% RSLogix 500 project LG01815_OriginalPLC_NoTags.RSS, saved by version 12.00.00.00 %
PROJECT "LVD4000"    % processor: MicroLogix 1400 %

PROGRAM FILES
  LAD 2   30 rungs
  LAD 3   3 rungs
  LAD 4   3 rungs
  LAD 5   3 rungs
  LAD 6   3 rungs
  LAD 7   8 rungs
  LAD 8   6 rungs
  LAD 10   21 rungs
  LAD 12   3 rungs
  LAD 14   12 rungs
  LAD 16   24 rungs
  LAD 18   5 rungs
  LAD 20   21 rungs
  LAD 22   2 rungs
  LAD 24   11 rungs
  LAD 26   14 rungs
  LAD 28   19 rungs
  LAD 30   6 rungs
  LAD 32   15 rungs
  LAD 34   20 rungs

DATA FILES
  O0 OUTPUT  6 elements
  I1 INPUT  8 elements
  S2 STATUS  66 elements
  B3 BINARY  256 elements
  T4 TIMER  32 elements
  C5 COUNTER  10 elements
  R6 CONTROL  9 elements
  N7 INTEGER  100 elements
  F8 FLOAT  30 elements
  B9   256 elements
  B11   256 elements
  B12   3 elements
  B14   256 elements
  B15   1 elements
  N16   14 elements
  N17   13 elements
  B18   256 elements
  F19   20 elements
  T20   13 elements
  R21   4 elements
  B22   256 elements
  B23   256 elements
  N24   128 elements
  B25   2 elements

LADDER 2
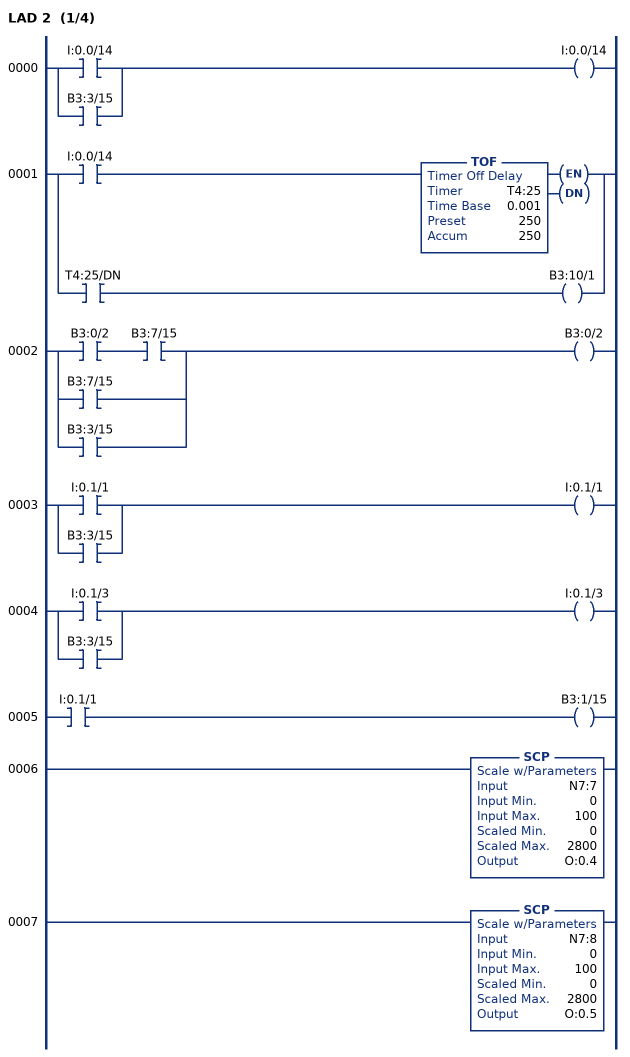
% Rung: 0 %
SOR BST XIC I:0.0/14 NXB XIC B3:3/15 BND OTE I:0.0/14 EOR
% Rung: 1 %
SOR BST XIC I:0.0/14 TOF T4:25 0.001 250 250 NXB XIC T4:25/DN OTE B3:10/1 BND EOR
% Rung: 2 %
SOR BST XIC B3:0/2 XIC B3:7/15 NXB XIC B3:7/15 NXB XIC B3:3/15 BND OTE B3:0/2 EOR
% Rung: 3 %
SOR BST XIC I:0.1/1 NXB XIC B3:3/15 BND OTE I:0.1/1 EOR
% Rung: 4 %
SOR BST XIC I:0.1/3 NXB XIC B3:3/15 BND OTE I:0.1/3 EOR
% Rung: 5 %
SOR XIC I:0.1/1 OTE B3:1/15 EOR
% Rung: 6 %
SOR SCP N7:7 0 100 0 2800 O:0.4 EOR
% Rung: 7 %
SOR SCP N7:8 0 100 0 2800 O:0.5 EOR

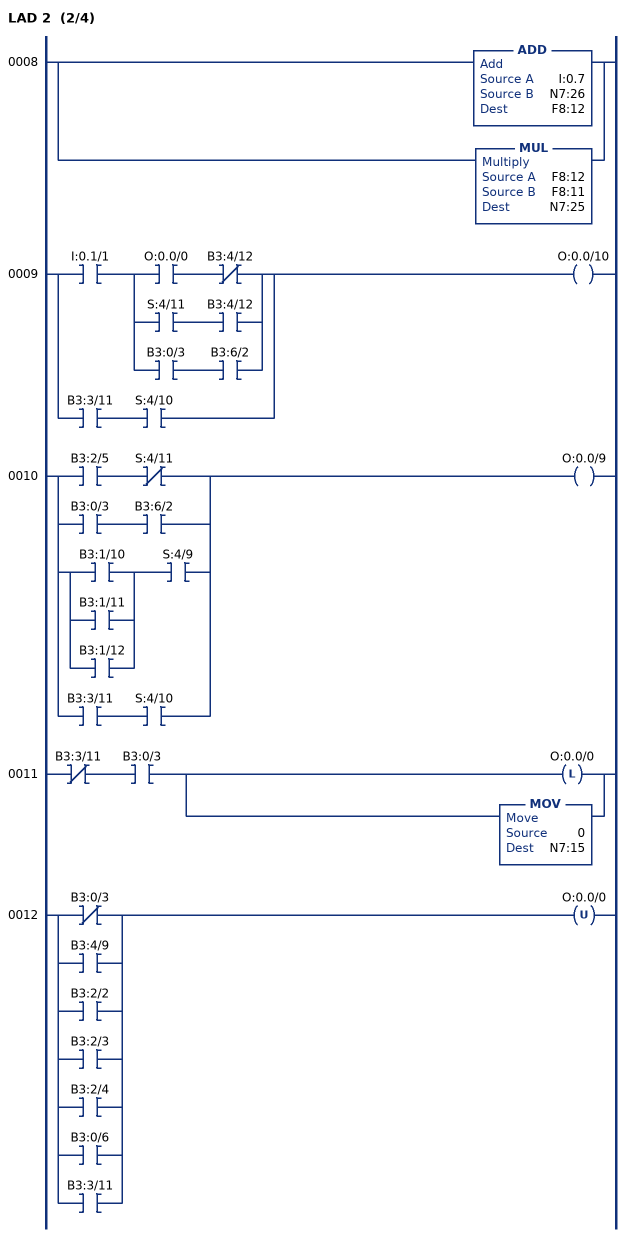
% Rung: 8 %
SOR BST ADD I:0.7 N7:26 F8:12 NXB MUL F8:12 F8:11 N7:25 BND EOR
% Rung: 9 %
SOR BST XIC I:0.1/1 BST XIC O:0.0/0 XIO B3:4/12 NXB XIC S:4/11 XIC B3:4/12 NXB XIC B3:0/3 XIC B3:6/2 BND NXB XIC B3:3/11 XIC S:4/10 BND OTE O:0.0/10 EOR
% Rung: 10 %
SOR BST BST XIC B3:2/5 XIO S:4/11 NXB XIC B3:0/3 XIC B3:6/2 NXB BST XIC B3:1/10 NXB XIC B3:1/11 NXB XIC B3:1/12 BND XIC S:4/9 BND NXB XIC B3:3/11 XIC S:4/10 BND OTE O:0.0/9 EOR
% Rung: 11 %
SOR XIO B3:3/11 XIC B3:0/3 BST OTL O:0.0/0 NXB MOV 0 N7:15 BND EOR
% Rung: 12 %
SOR BST XIO B3:0/3 NXB XIC B3:4/9 NXB XIC B3:2/2 NXB XIC B3:2/3 NXB XIC B3:2/4 NXB XIC B3:0/6 NXB XIC B3:3/11 BND OTU O:0.0/0 EOR

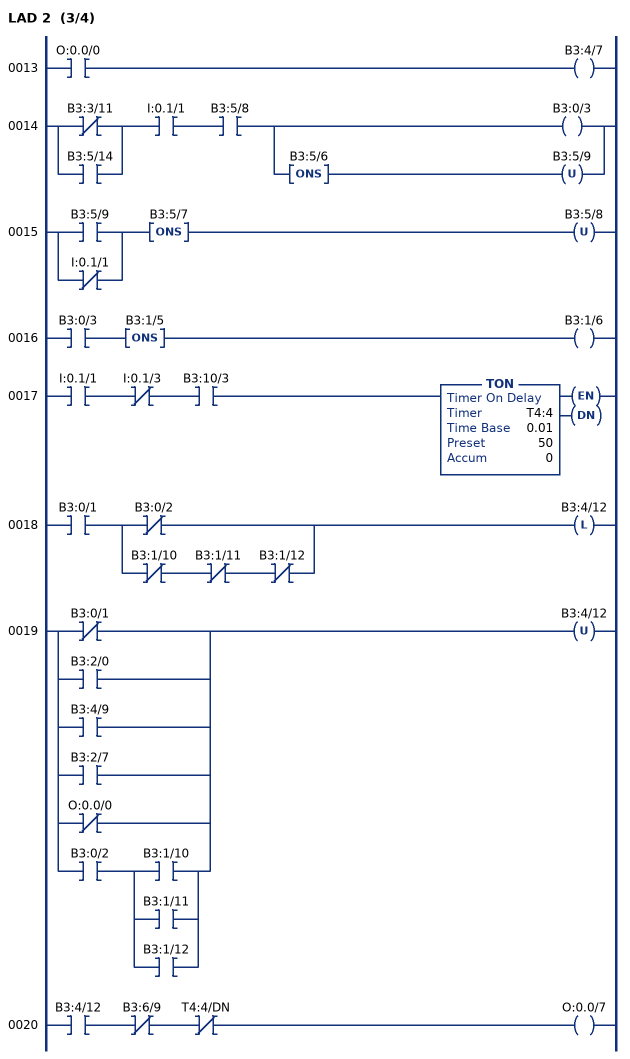
% Rung: 13 %
SOR XIC O:0.0/0 OTE B3:4/7 EOR
% Rung: 14 %
SOR BST XIO B3:3/11 NXB XIC B3:5/14 BND XIC I:0.1/1 XIC B3:5/8 BST OTE B3:0/3 NXB ONS B3:5/6 OTU B3:5/9 BND EOR
% Rung: 15 %
SOR BST XIC B3:5/9 NXB XIO I:0.1/1 BND ONS B3:5/7 OTU B3:5/8 EOR
% Rung: 16 %
SOR XIC B3:0/3 ONS B3:1/5 OTE B3:1/6 EOR
% Rung: 17 %
SOR XIC I:0.1/1 XIO I:0.1/3 XIC B3:10/3 TON T4:4 0.01 50 0 EOR
% Rung: 18 %
SOR XIC B3:0/1 BST XIO B3:0/2 NXB XIO B3:1/10 XIO B3:1/11 XIO B3:1/12 BND OTL B3:4/12 EOR
% Rung: 19 %
SOR BST XIO B3:0/1 NXB XIC B3:2/0 NXB XIC B3:4/9 NXB XIC B3:2/7 NXB XIO O:0.0/0 NXB XIC B3:0/2 BST XIC B3:1/10 NXB XIC B3:1/11 NXB XIC B3:1/12 BND BND OTU B3:4/12 EOR
% Rung: 20 %
SOR XIC B3:4/12 XIO B3:6/9 XIO T4:4/DN OTE O:0.0/7 EOR

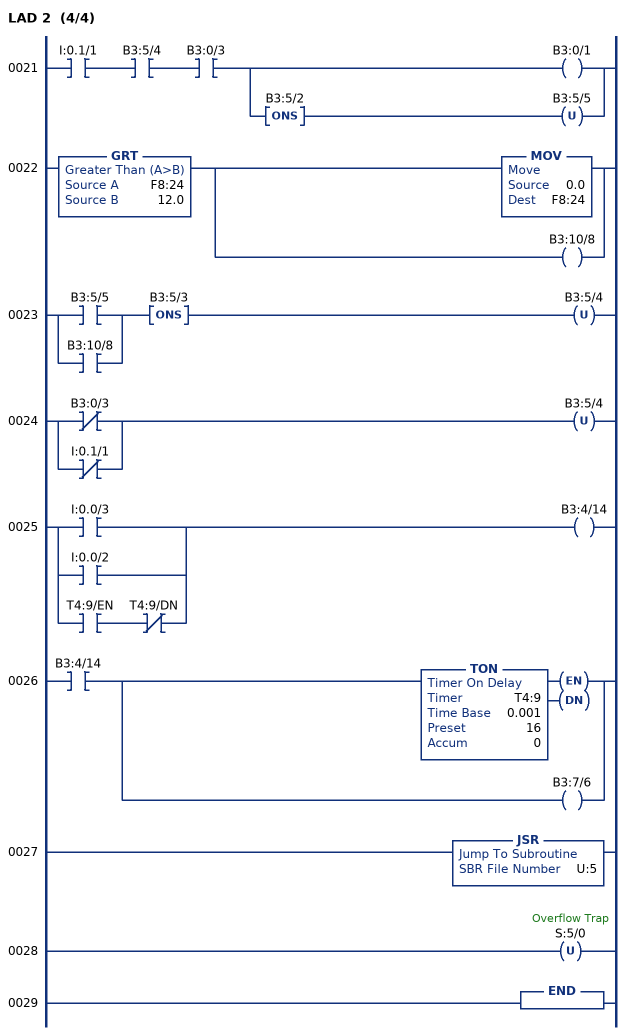
% Rung: 21 %
SOR XIC I:0.1/1 XIC B3:5/4 XIC B3:0/3 BST OTE B3:0/1 NXB ONS B3:5/2 OTU B3:5/5 BND EOR
% Rung: 22 %
SOR GRT F8:24 12.0 BST MOV 0.0 F8:24 NXB OTE B3:10/8 BND EOR
% Rung: 23 %
SOR BST XIC B3:5/5 NXB XIC B3:10/8 BND ONS B3:5/3 OTU B3:5/4 EOR
% Rung: 24 %
SOR BST XIO B3:0/3 NXB XIO I:0.1/1 BND OTU B3:5/4 EOR
% Rung: 25 %
SOR BST XIC I:0.0/3 NXB XIC I:0.0/2 NXB XIC T4:9/EN XIO T4:9/DN BND OTE B3:4/14 EOR
% Rung: 26 %
SOR XIC B3:4/14 BST TON T4:9 0.001 16 0 NXB OTE B3:7/6 BND EOR
% Rung: 27 %
SOR JSR U:5 EOR
% Rung: 28 %
SOR OTU S:5/0 EOR
%   S:5/0  "Overflow Trap" %
% Rung: 29 %
SOR END EOR

LADDER 3
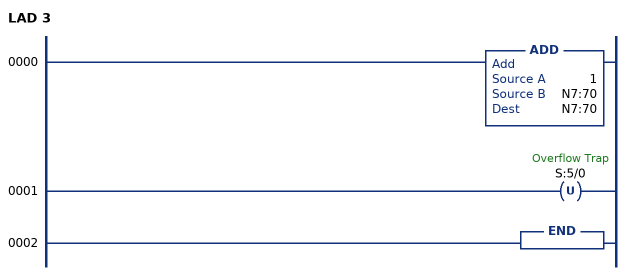
% Rung: 0 %
SOR ADD 1 N7:70 N7:70 EOR
% Rung: 1 %
SOR OTU S:5/0 EOR
%   S:5/0  "Overflow Trap" %
% Rung: 2 %
SOR END EOR

LADDER 4
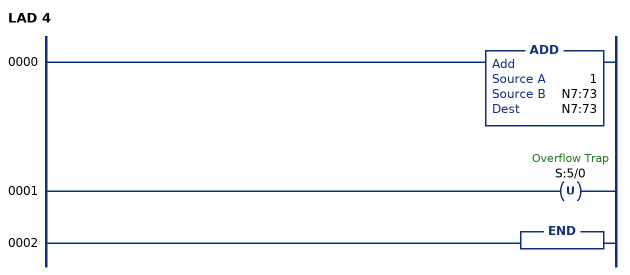
% Rung: 0 %
SOR ADD 1 N7:73 N7:73 EOR
% Rung: 1 %
SOR OTU S:5/0 EOR
%   S:5/0  "Overflow Trap" %
% Rung: 2 %
SOR END EOR

LADDER 5
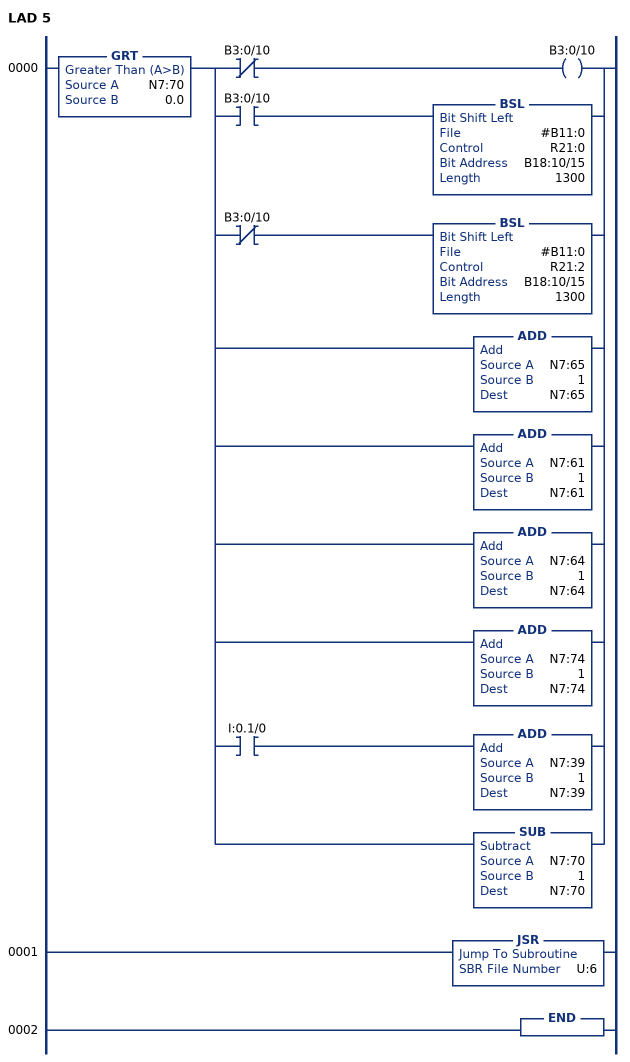
% Rung: 0 %
SOR GRT N7:70 0.0 BST XIO B3:0/10 OTE B3:0/10 NXB XIC B3:0/10 BSL #B11:0 R21:0 B18:10/15 1300 NXB XIO B3:0/10 BSL #B11:0 R21:2 B18:10/15 1300 NXB ADD N7:65 1 N7:65 NXB ADD N7:61 1 N7:61 NXB ADD N7:64 1 N7:64 NXB ADD N7:74 1 N7:74 NXB XIC I:0.1/0 ADD N7:39 1 N7:39 NXB SUB N7:70 1 N7:70 BND EOR
% Rung: 1 %
SOR JSR U:6 EOR
% Rung: 2 %
SOR END EOR

LADDER 6
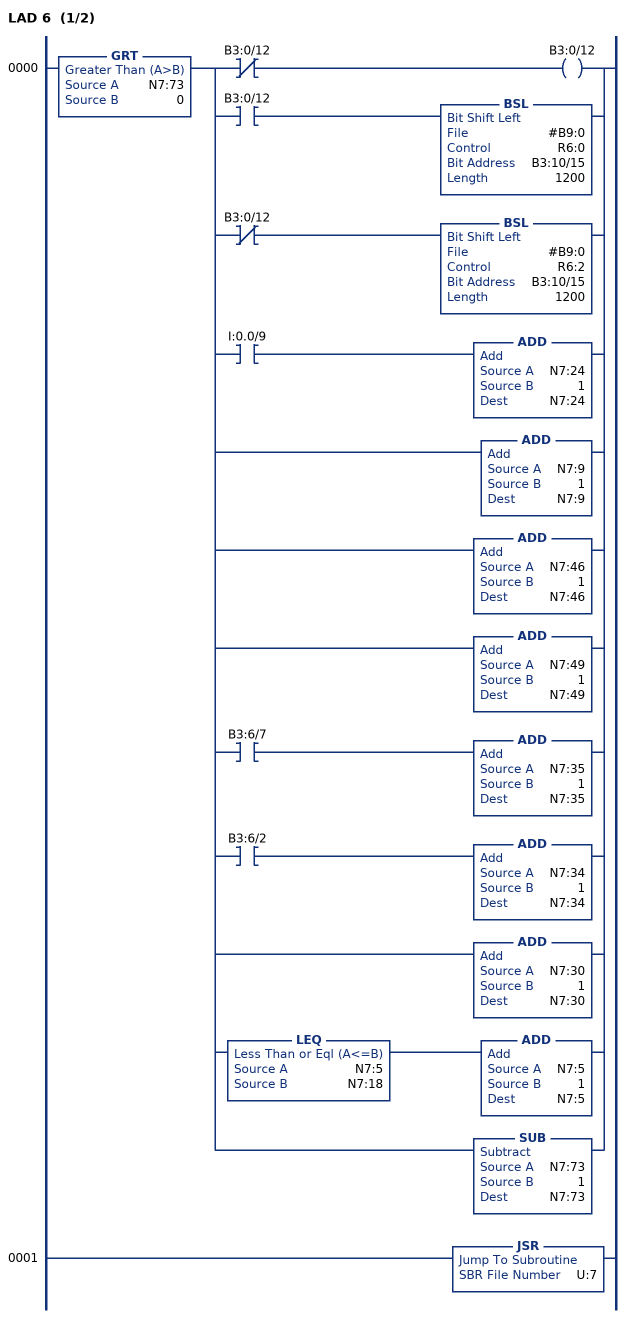
% Rung: 0 %
SOR GRT N7:73 0 BST XIO B3:0/12 OTE B3:0/12 NXB XIC B3:0/12 BSL #B9:0 R6:0 B3:10/15 1200 NXB XIO B3:0/12 BSL #B9:0 R6:2 B3:10/15 1200 NXB XIC I:0.0/9 ADD N7:24 1 N7:24 NXB ADD N7:9 1 N7:9 NXB ADD N7:46 1 N7:46 NXB ADD N7:49 1 N7:49 NXB XIC B3:6/7 ADD N7:35 1 N7:35 NXB XIC B3:6/2 ADD N7:34 1 N7:34 NXB ADD N7:30 1 N7:30 NXB LEQ N7:5 N7:18 ADD N7:5 1 N7:5 NXB SUB N7:73 1 N7:73 BND EOR
% Rung: 1 %
SOR JSR U:7 EOR

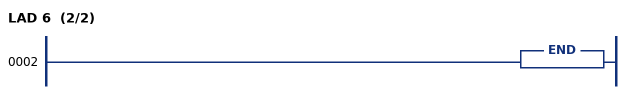
% Rung: 2 %
SOR END EOR

LADDER 7
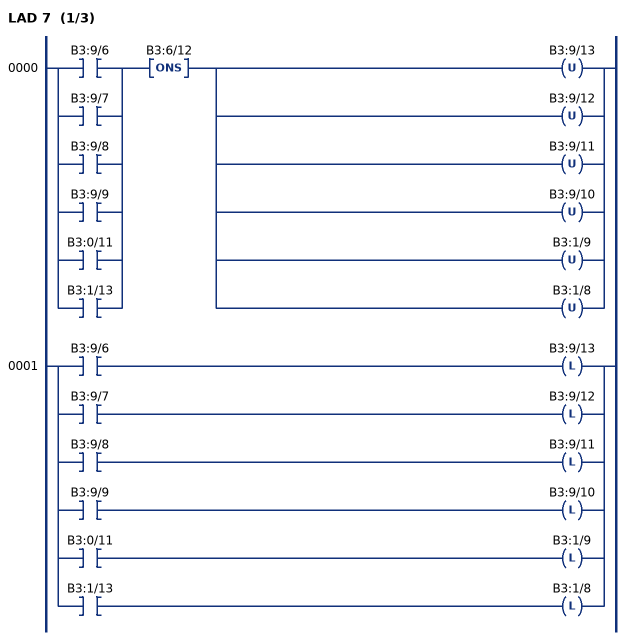
% Rung: 0 %
SOR BST XIC B3:9/6 NXB XIC B3:9/7 NXB XIC B3:9/8 NXB XIC B3:9/9 NXB XIC B3:0/11 NXB XIC B3:1/13 BND ONS B3:6/12 BST OTU B3:9/13 NXB OTU B3:9/12 NXB OTU B3:9/11 NXB OTU B3:9/10 NXB OTU B3:1/9 NXB OTU B3:1/8 BND EOR
% Rung: 1 %
SOR BST XIC B3:9/6 OTL B3:9/13 NXB XIC B3:9/7 OTL B3:9/12 NXB XIC B3:9/8 OTL B3:9/11 NXB XIC B3:9/9 OTL B3:9/10 NXB XIC B3:0/11 OTL B3:1/9 NXB XIC B3:1/13 OTL B3:1/8 BND EOR

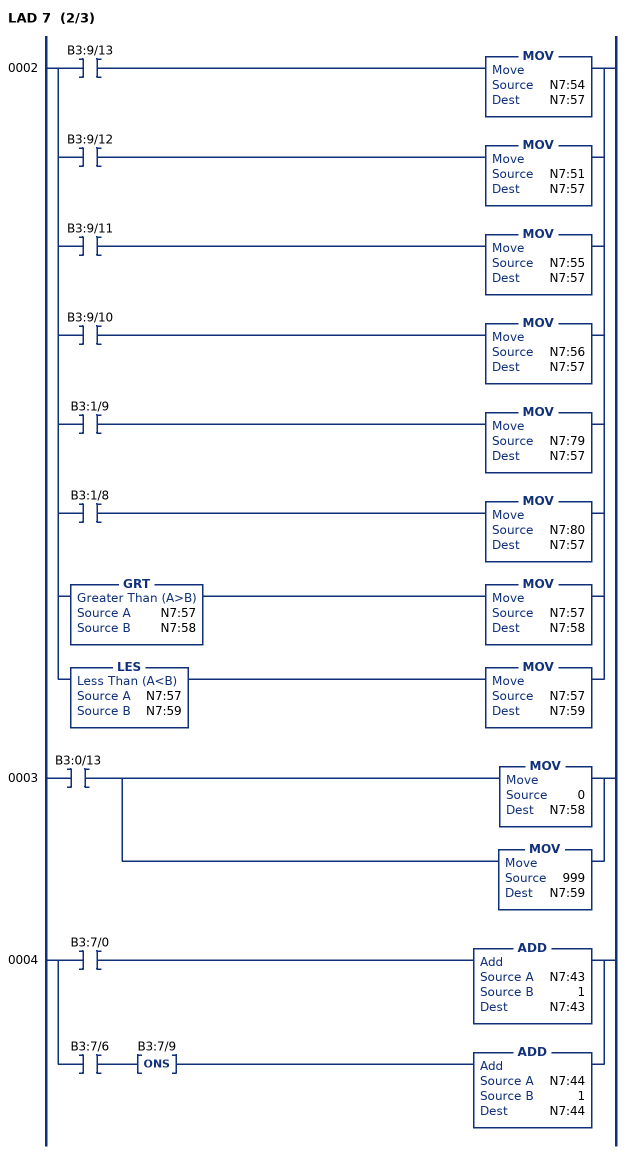
% Rung: 2 %
SOR BST XIC B3:9/13 MOV N7:54 N7:57 NXB XIC B3:9/12 MOV N7:51 N7:57 NXB XIC B3:9/11 MOV N7:55 N7:57 NXB XIC B3:9/10 MOV N7:56 N7:57 NXB XIC B3:1/9 MOV N7:79 N7:57 NXB XIC B3:1/8 MOV N7:80 N7:57 NXB GRT N7:57 N7:58 MOV N7:57 N7:58 NXB LES N7:57 N7:59 MOV N7:57 N7:59 BND EOR
% Rung: 3 %
SOR XIC B3:0/13 BST MOV 0 N7:58 NXB MOV 999 N7:59 BND EOR
% Rung: 4 %
SOR BST XIC B3:7/0 ADD N7:43 1 N7:43 NXB XIC B3:7/6 ONS B3:7/9 ADD N7:44 1 N7:44 BND EOR

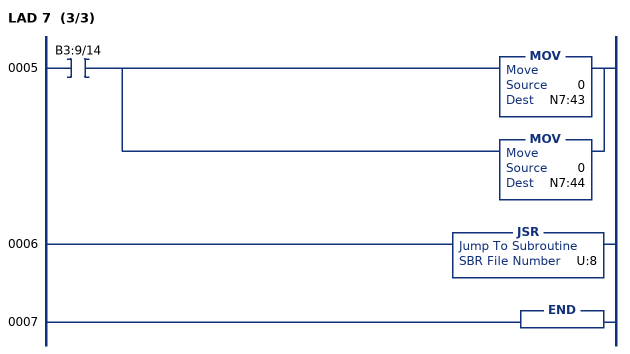
% Rung: 5 %
SOR XIC B3:9/14 BST MOV 0 N7:43 NXB MOV 0 N7:44 BND EOR
% Rung: 6 %
SOR JSR U:8 EOR
% Rung: 7 %
SOR END EOR

LADDER 8
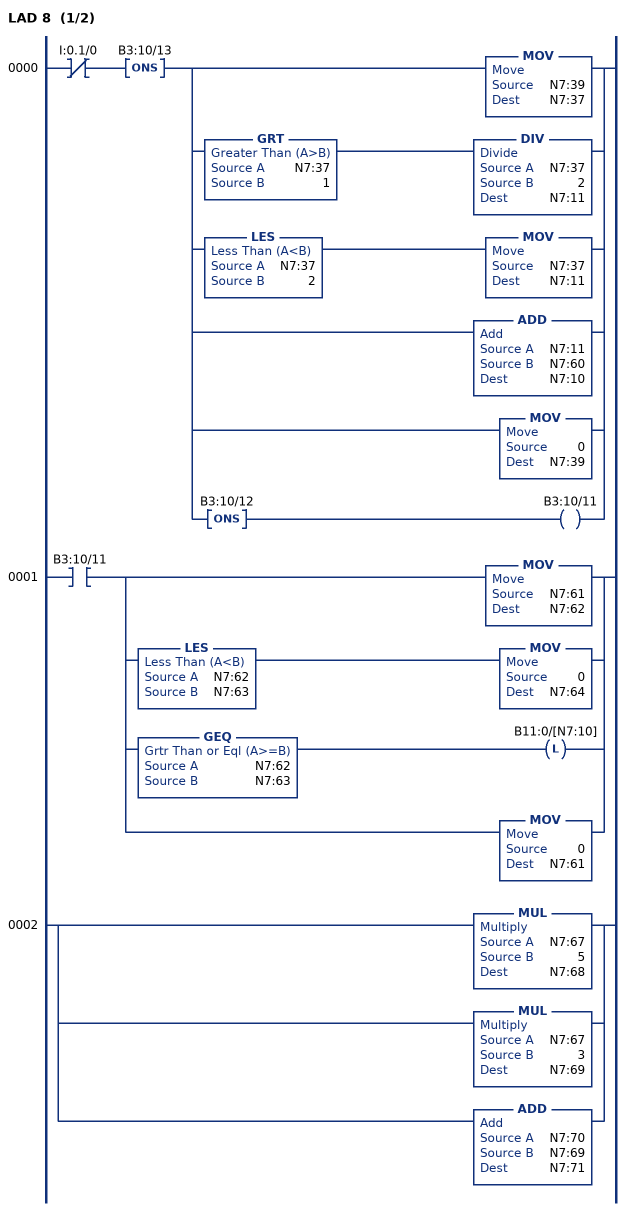
% Rung: 0 %
SOR XIO I:0.1/0 ONS B3:10/13 BST MOV N7:39 N7:37 NXB GRT N7:37 1 DIV N7:37 2 N7:11 NXB LES N7:37 2 MOV N7:37 N7:11 NXB ADD N7:11 N7:60 N7:10 NXB MOV 0 N7:39 NXB ONS B3:10/12 OTE B3:10/11 BND EOR
% Rung: 1 %
SOR XIC B3:10/11 BST MOV N7:61 N7:62 NXB LES N7:62 N7:63 MOV 0 N7:64 NXB GEQ N7:62 N7:63 OTL B11:0/[N7:10] NXB MOV 0 N7:61 BND EOR
% Rung: 2 %
SOR BST MUL N7:67 5 N7:68 NXB MUL N7:67 3 N7:69 NXB ADD N7:70 N7:69 N7:71 BND EOR

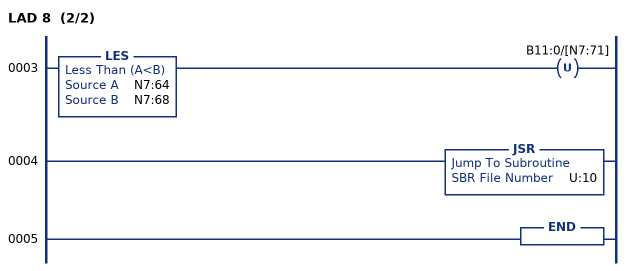
% Rung: 3 %
SOR LES N7:64 N7:68 OTU B11:0/[N7:71] EOR
% Rung: 4 %
SOR JSR U:10 EOR
% Rung: 5 %
SOR END EOR

LADDER 10
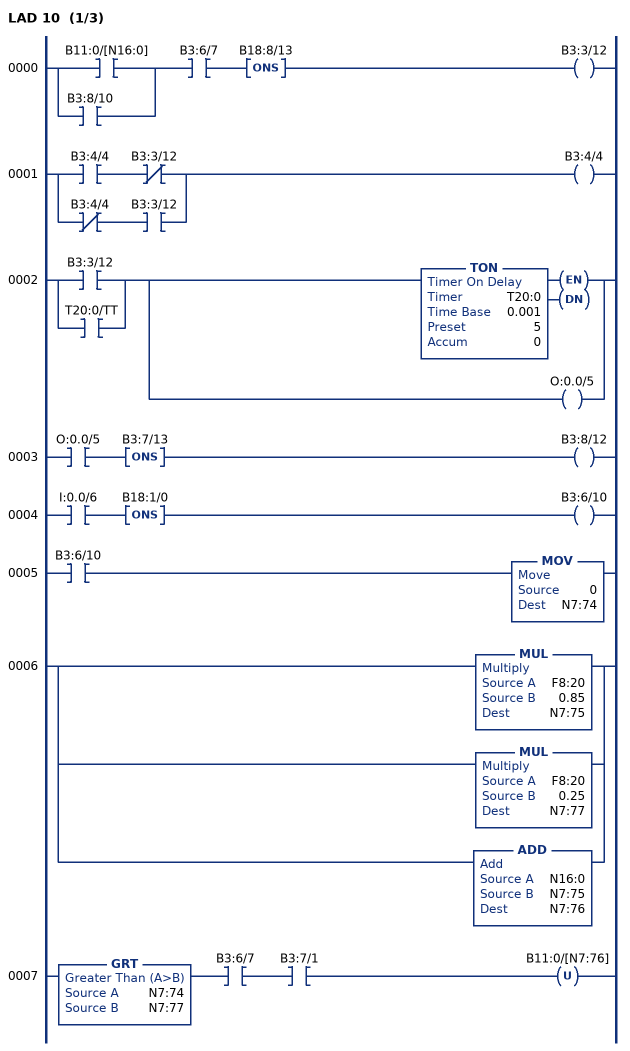
% Rung: 0 %
SOR BST XIC B11:0/[N16:0] NXB XIC B3:8/10 BND XIC B3:6/7 ONS B18:8/13 OTE B3:3/12 EOR
% Rung: 1 %
SOR BST XIC B3:4/4 XIO B3:3/12 NXB XIO B3:4/4 XIC B3:3/12 BND OTE B3:4/4 EOR
% Rung: 2 %
SOR BST XIC B3:3/12 NXB XIC T20:0/TT BND BST TON T20:0 0.001 5 0 NXB OTE O:0.0/5 BND EOR
% Rung: 3 %
SOR XIC O:0.0/5 ONS B3:7/13 OTE B3:8/12 EOR
% Rung: 4 %
SOR XIC I:0.0/6 ONS B18:1/0 OTE B3:6/10 EOR
% Rung: 5 %
SOR XIC B3:6/10 MOV 0 N7:74 EOR
% Rung: 6 %
SOR BST MUL F8:20 0.85 N7:75 NXB MUL F8:20 0.25 N7:77 NXB ADD N16:0 N7:75 N7:76 BND EOR
% Rung: 7 %
SOR GRT N7:74 N7:77 XIC B3:6/7 XIC B3:7/1 OTU B11:0/[N7:76] EOR

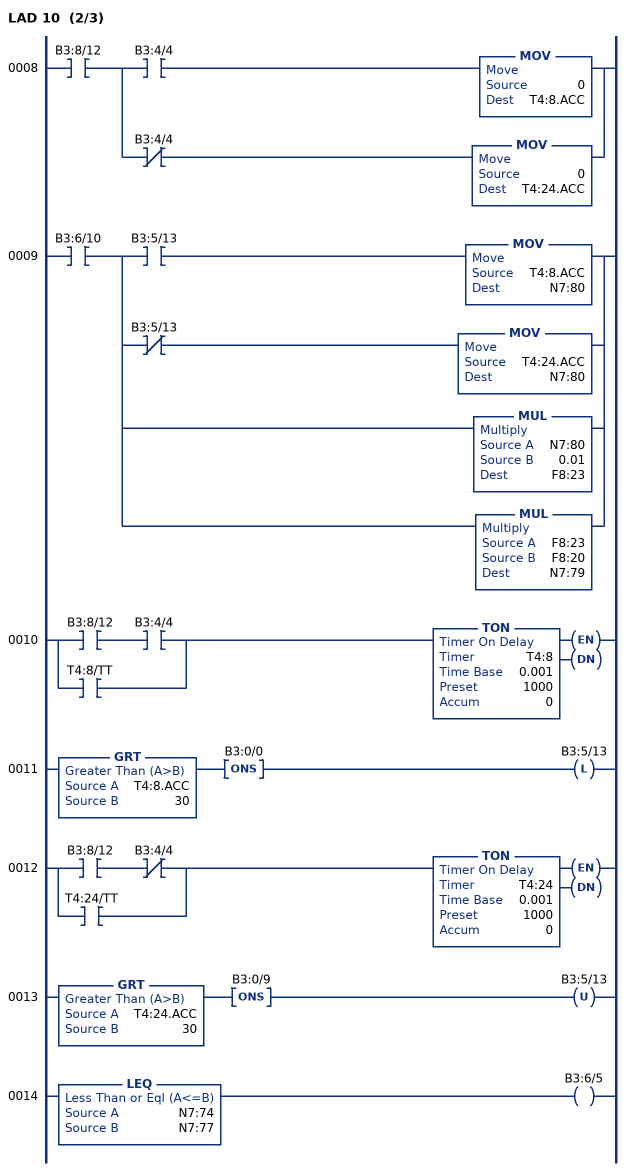
% Rung: 8 %
SOR XIC B3:8/12 BST XIC B3:4/4 MOV 0 T4:8.ACC NXB XIO B3:4/4 MOV 0 T4:24.ACC BND EOR
% Rung: 9 %
SOR XIC B3:6/10 BST XIC B3:5/13 MOV T4:8.ACC N7:80 NXB XIO B3:5/13 MOV T4:24.ACC N7:80 NXB MUL N7:80 0.01 F8:23 NXB MUL F8:23 F8:20 N7:79 BND EOR
% Rung: 10 %
SOR BST XIC B3:8/12 XIC B3:4/4 NXB XIC T4:8/TT BND TON T4:8 0.001 1000 0 EOR
% Rung: 11 %
SOR GRT T4:8.ACC 30 ONS B3:0/0 OTL B3:5/13 EOR
% Rung: 12 %
SOR BST XIC B3:8/12 XIO B3:4/4 NXB XIC T4:24/TT BND TON T4:24 0.001 1000 0 EOR
% Rung: 13 %
SOR GRT T4:24.ACC 30 ONS B3:0/9 OTU B3:5/13 EOR
% Rung: 14 %
SOR LEQ N7:74 N7:77 OTE B3:6/5 EOR

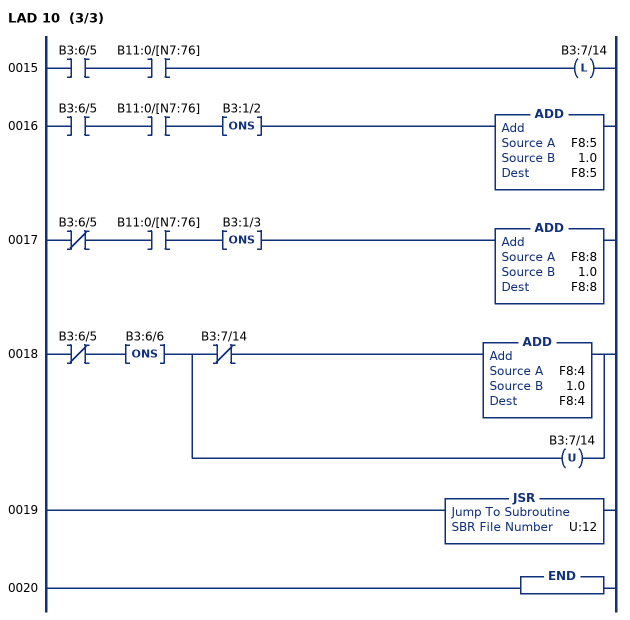
% Rung: 15 %
SOR XIC B3:6/5 XIC B11:0/[N7:76] OTL B3:7/14 EOR
% Rung: 16 %
SOR XIC B3:6/5 XIC B11:0/[N7:76] ONS B3:1/2 ADD F8:5 1.0 F8:5 EOR
% Rung: 17 %
SOR XIO B3:6/5 XIC B11:0/[N7:76] ONS B3:1/3 ADD F8:8 1.0 F8:8 EOR
% Rung: 18 %
SOR XIO B3:6/5 ONS B3:6/6 BST XIO B3:7/14 ADD F8:4 1.0 F8:4 NXB OTU B3:7/14 BND EOR
% Rung: 19 %
SOR JSR U:12 EOR
% Rung: 20 %
SOR END EOR

LADDER 12
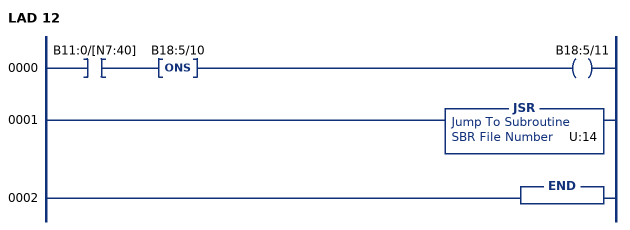
% Rung: 0 %
SOR XIC B11:0/[N7:40] ONS B18:5/10 OTE B18:5/11 EOR
% Rung: 1 %
SOR JSR U:14 EOR
% Rung: 2 %
SOR END EOR

LADDER 14
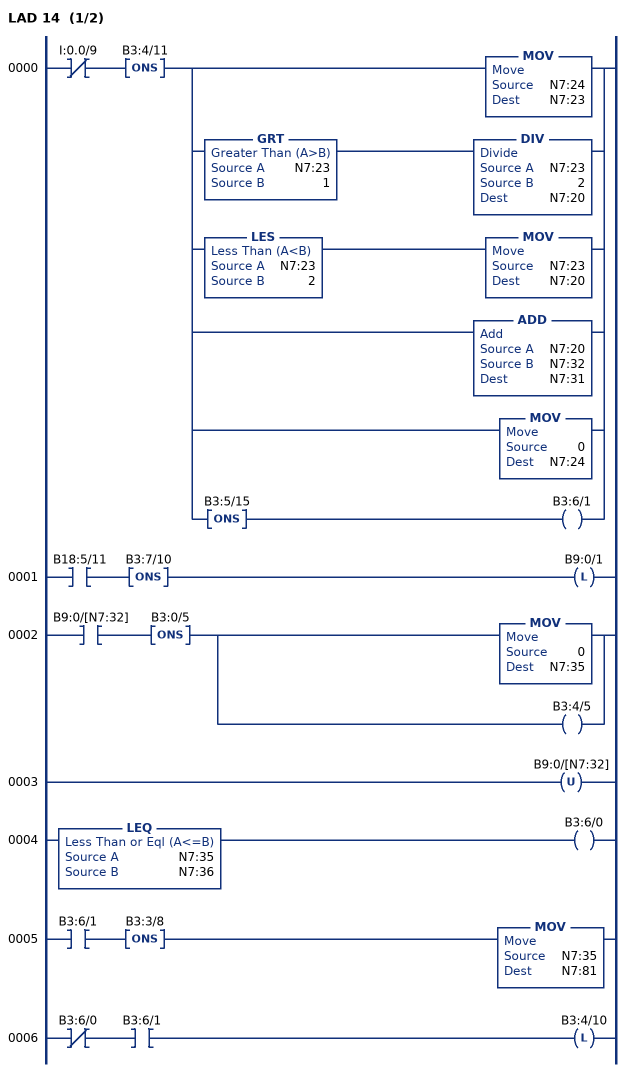
% Rung: 0 %
SOR XIO I:0.0/9 ONS B3:4/11 BST MOV N7:24 N7:23 NXB GRT N7:23 1 DIV N7:23 2 N7:20 NXB LES N7:23 2 MOV N7:23 N7:20 NXB ADD N7:20 N7:32 N7:31 NXB MOV 0 N7:24 NXB ONS B3:5/15 OTE B3:6/1 BND EOR
% Rung: 1 %
SOR XIC B18:5/11 ONS B3:7/10 OTL B9:0/1 EOR
% Rung: 2 %
SOR XIC B9:0/[N7:32] ONS B3:0/5 BST MOV 0 N7:35 NXB OTE B3:4/5 BND EOR
% Rung: 3 %
SOR OTU B9:0/[N7:32] EOR
% Rung: 4 %
SOR LEQ N7:35 N7:36 OTE B3:6/0 EOR
% Rung: 5 %
SOR XIC B3:6/1 ONS B3:3/8 MOV N7:35 N7:81 EOR
% Rung: 6 %
SOR XIO B3:6/0 XIC B3:6/1 OTL B3:4/10 EOR

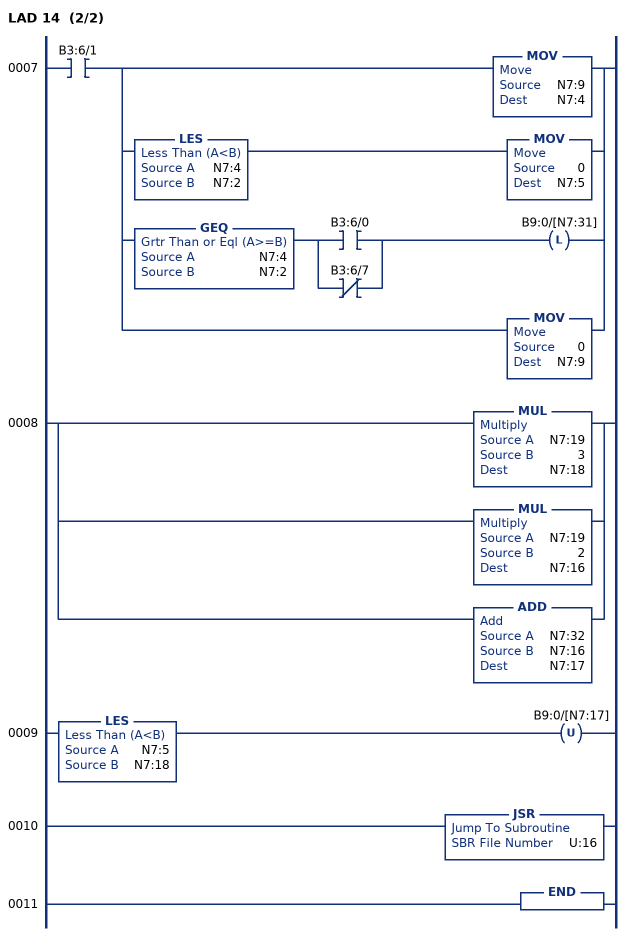
% Rung: 7 %
SOR XIC B3:6/1 BST MOV N7:9 N7:4 NXB LES N7:4 N7:2 MOV 0 N7:5 NXB GEQ N7:4 N7:2 BST XIC B3:6/0 NXB XIO B3:6/7 BND OTL B9:0/[N7:31] NXB MOV 0 N7:9 BND EOR
% Rung: 8 %
SOR BST MUL N7:19 3 N7:18 NXB MUL N7:19 2 N7:16 NXB ADD N7:32 N7:16 N7:17 BND EOR
% Rung: 9 %
SOR LES N7:5 N7:18 OTU B9:0/[N7:17] EOR
% Rung: 10 %
SOR JSR U:16 EOR
% Rung: 11 %
SOR END EOR

LADDER 16
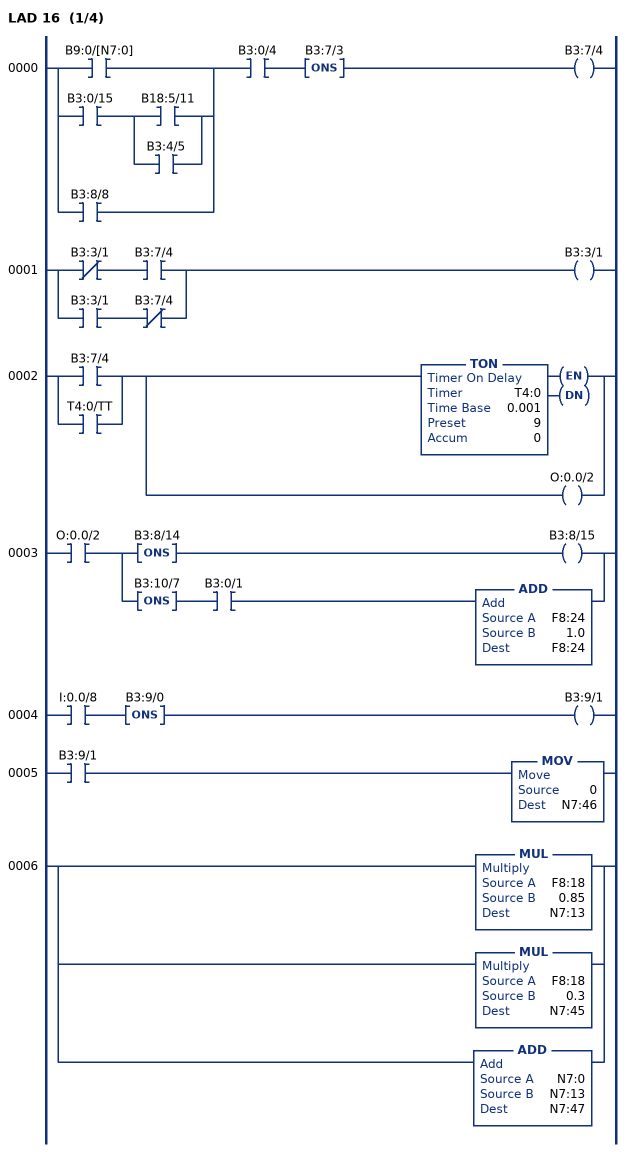
% Rung: 0 %
SOR BST XIC B9:0/[N7:0] NXB XIC B3:0/15 BST XIC B18:5/11 NXB XIC B3:4/5 BND NXB XIC B3:8/8 BND XIC B3:0/4 ONS B3:7/3 OTE B3:7/4 EOR
% Rung: 1 %
SOR BST XIO B3:3/1 XIC B3:7/4 NXB XIC B3:3/1 XIO B3:7/4 BND OTE B3:3/1 EOR
% Rung: 2 %
SOR BST XIC B3:7/4 NXB XIC T4:0/TT BND BST TON T4:0 0.001 9 0 NXB OTE O:0.0/2 BND EOR
% Rung: 3 %
SOR XIC O:0.0/2 BST ONS B3:8/14 OTE B3:8/15 NXB ONS B3:10/7 XIC B3:0/1 ADD F8:24 1.0 F8:24 BND EOR
% Rung: 4 %
SOR XIC I:0.0/8 ONS B3:9/0 OTE B3:9/1 EOR
% Rung: 5 %
SOR XIC B3:9/1 MOV 0 N7:46 EOR
% Rung: 6 %
SOR BST MUL F8:18 0.85 N7:13 NXB MUL F8:18 0.3 N7:45 NXB ADD N7:0 N7:13 N7:47 BND EOR

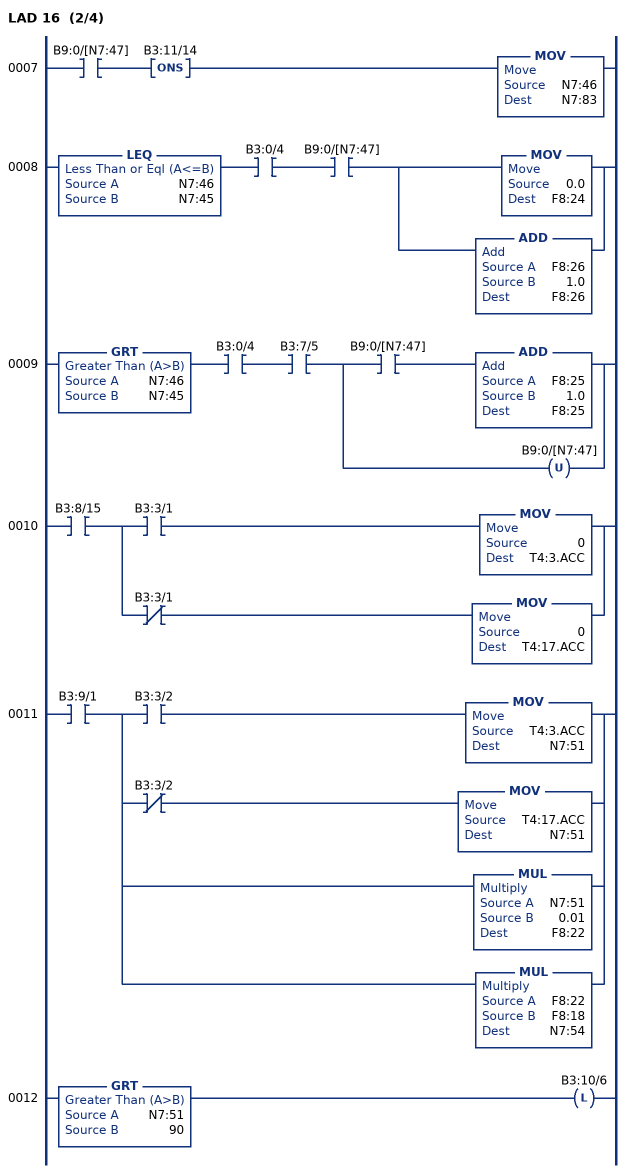
% Rung: 7 %
SOR XIC B9:0/[N7:47] ONS B3:11/14 MOV N7:46 N7:83 EOR
% Rung: 8 %
SOR LEQ N7:46 N7:45 XIC B3:0/4 XIC B9:0/[N7:47] BST MOV 0.0 F8:24 NXB ADD F8:26 1.0 F8:26 BND EOR
% Rung: 9 %
SOR GRT N7:46 N7:45 XIC B3:0/4 XIC B3:7/5 BST XIC B9:0/[N7:47] ADD F8:25 1.0 F8:25 NXB OTU B9:0/[N7:47] BND EOR
% Rung: 10 %
SOR XIC B3:8/15 BST XIC B3:3/1 MOV 0 T4:3.ACC NXB XIO B3:3/1 MOV 0 T4:17.ACC BND EOR
% Rung: 11 %
SOR XIC B3:9/1 BST XIC B3:3/2 MOV T4:3.ACC N7:51 NXB XIO B3:3/2 MOV T4:17.ACC N7:51 NXB MUL N7:51 0.01 F8:22 NXB MUL F8:22 F8:18 N7:54 BND EOR
% Rung: 12 %
SOR GRT N7:51 90 OTL B3:10/6 EOR

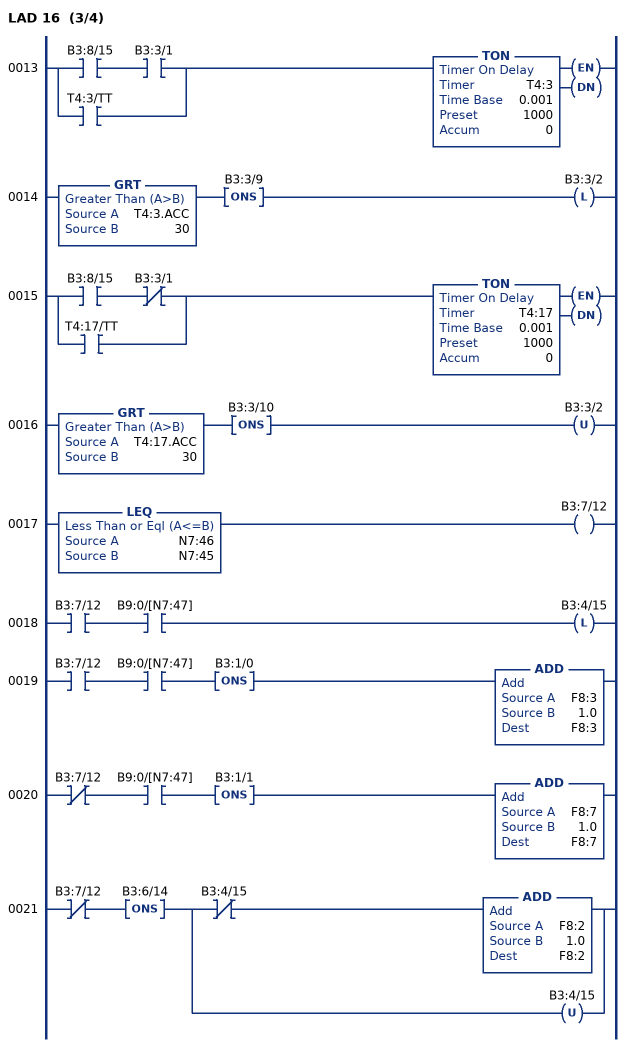
% Rung: 13 %
SOR BST XIC B3:8/15 XIC B3:3/1 NXB XIC T4:3/TT BND TON T4:3 0.001 1000 0 EOR
% Rung: 14 %
SOR GRT T4:3.ACC 30 ONS B3:3/9 OTL B3:3/2 EOR
% Rung: 15 %
SOR BST XIC B3:8/15 XIO B3:3/1 NXB XIC T4:17/TT BND TON T4:17 0.001 1000 0 EOR
% Rung: 16 %
SOR GRT T4:17.ACC 30 ONS B3:3/10 OTU B3:3/2 EOR
% Rung: 17 %
SOR LEQ N7:46 N7:45 OTE B3:7/12 EOR
% Rung: 18 %
SOR XIC B3:7/12 XIC B9:0/[N7:47] OTL B3:4/15 EOR
% Rung: 19 %
SOR XIC B3:7/12 XIC B9:0/[N7:47] ONS B3:1/0 ADD F8:3 1.0 F8:3 EOR
% Rung: 20 %
SOR XIO B3:7/12 XIC B9:0/[N7:47] ONS B3:1/1 ADD F8:7 1.0 F8:7 EOR
% Rung: 21 %
SOR XIO B3:7/12 ONS B3:6/14 BST XIO B3:4/15 ADD F8:2 1.0 F8:2 NXB OTU B3:4/15 BND EOR

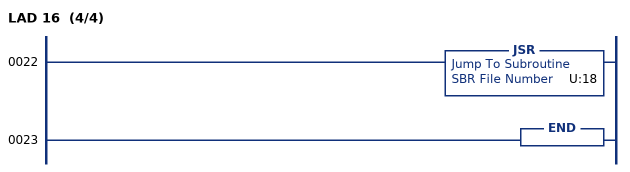
% Rung: 22 %
SOR JSR U:18 EOR
% Rung: 23 %
SOR END EOR

LADDER 18
